// TIA Portal project "Soru9" (V15)

(* hardware
DEVICE "S7-1200 station_1"  S7-1200 Station
   slot 0: "Rack_0"  S7-1200 Rack  Rack  V1.0
   slot 1: "PLC_1"  CPU 1214C DC/DC/DC  6ES7 214-1AG40-0XB0  V4.2
*)

// ===== PLC "PLC_1"  CPU 1214C DC/DC/DC =====

VAR_GLOBAL   // PLC tag table "Default tag table"
   "Baslat" AT %I0.0 : Bool;
   "Durdur" AT %I0.1 : Bool;
   "Termik_Anahtar_Bant_1" AT %I0.2 : Bool;
   "Termik_Anahtar_Bant_2" AT %I0.3 : Bool;
   "Termik_Anahtar_Bant_3" AT %I0.4 : Bool;
   "Bant_1" AT %Q0.0 : Bool;
   "Bant_2" AT %Q0.1 : Bool;
   "Bant_3" AT %Q0.2 : Bool;
   "Aşırı_akım" AT %I0.5 : Bool;
END_VAR

// folder: System blocks/Program resources

DATA_BLOCK "Baslat_Time"   // DB2
{ S7_Optimized_Access := 'TRUE' }
AUTHOR : Simatic
FAMILY : IEC
NAME : IEC_TMR
VERSION : 1.0
// stored: InstanceOfName IEC_TIMER
"IEC_TIMER"
BEGIN
END_DATA_BLOCK

DATA_BLOCK "Dudur_Timer"   // DB3
{ S7_Optimized_Access := 'TRUE' }
AUTHOR : Simatic
FAMILY : IEC
NAME : IEC_TMR
VERSION : 1.0
// stored: InstanceOfName IEC_TIMER
"IEC_TIMER"
BEGIN
END_DATA_BLOCK

// folder: (top level)

ORGANIZATION_BLOCK "Main"   // OB1, LAD, ProgramCycle
TITLE = "Main Program Sweep (Cycle)"
{ S7_Optimized_Access := 'TRUE' }
VERSION : 0.1
   VAR_INPUT
      Initial_Call : Bool;   // Initial call of this OB
      Remanence : Bool;   // =True, if remanent data are available
   END_VAR
BEGIN

REGION Network 1: Baslama için Zaman bölümü
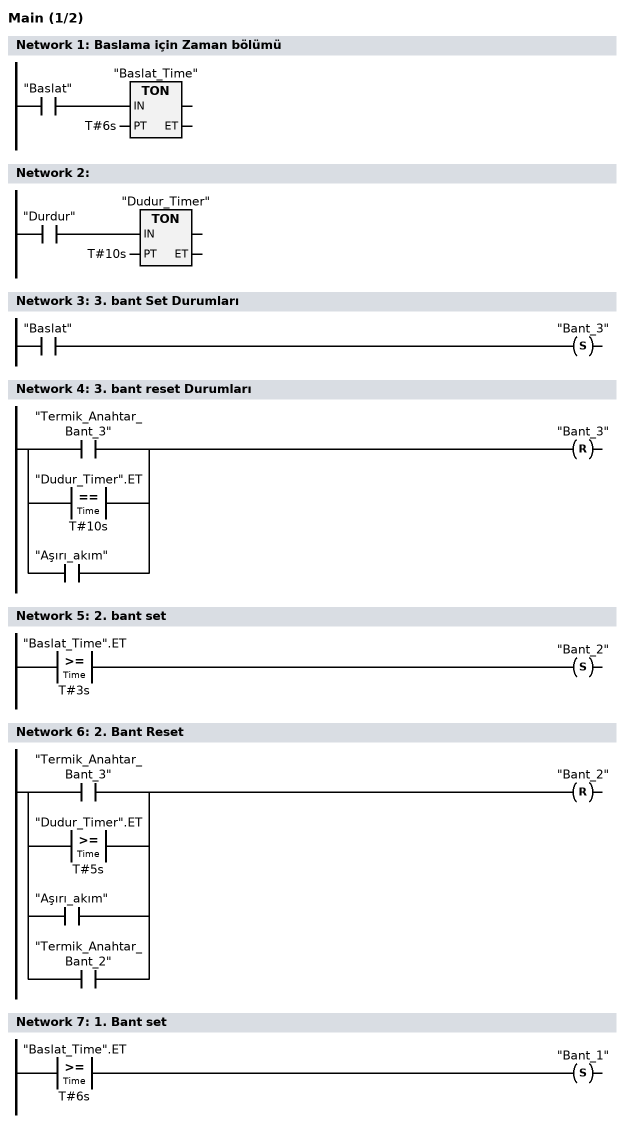
   "Baslat_Time".TON(IN := "Baslat", PT := T#6s);
END_REGION

REGION Network 2
   "Dudur_Timer".TON(IN := "Durdur", PT := T#10s);
END_REGION

REGION Network 3: 3. bant Set Durumları
   RUNG wire#powerrail
      Contact( "Baslat" )
      S_Coil( "Bant_3" )
   END_RUNG
   // the same network as SCL:
   IF "Baslat" THEN "Bant_3" := TRUE; END_IF;
END_REGION

REGION Network 4: 3. bant reset Durumları
   RUNG wire#powerrail
      Contact( "Termik_Anahtar_Bant_3" )
      wire#w1
      R_Coil( "Bant_3" )
   END_RUNG
   RUNG wire#powerrail
      { S7_Templates := "SrcType := Time" } EQ_Contact(in1 := "Dudur_Timer".ET, in2 := T#10s)
   END_RUNG wire#w1
   RUNG wire#powerrail
      Contact( "Aşırı_akım" )
   END_RUNG wire#w1
   // the same network as SCL:
   IF "Termik_Anahtar_Bant_3" OR ("Dudur_Timer".ET = T#10s) OR "Aşırı_akım" THEN "Bant_3" := FALSE; END_IF;
END_REGION

REGION Network 5: 2. bant set
   RUNG wire#powerrail
      { S7_Templates := "SrcType := Time" } GE_Contact(in1 := "Baslat_Time".ET, in2 := T#3s)
      S_Coil( "Bant_2" )
   END_RUNG
   // the same network as SCL:
   IF "Baslat_Time".ET >= T#3s THEN "Bant_2" := TRUE; END_IF;
END_REGION

REGION Network 6: 2. Bant Reset
   RUNG wire#powerrail
      Contact( "Termik_Anahtar_Bant_3" )
      wire#w1
      R_Coil( "Bant_2" )
   END_RUNG
   RUNG wire#powerrail
      { S7_Templates := "SrcType := Time" } GE_Contact(in1 := "Dudur_Timer".ET, in2 := T#5s)
   END_RUNG wire#w1
   RUNG wire#powerrail
      Contact( "Aşırı_akım" )
   END_RUNG wire#w1
   RUNG wire#powerrail
      Contact( "Termik_Anahtar_Bant_2" )
   END_RUNG wire#w1
   // the same network as SCL:
   IF "Termik_Anahtar_Bant_3" OR ("Dudur_Timer".ET >= T#5s) OR "Aşırı_akım" OR "Termik_Anahtar_Bant_2" THEN
       "Bant_2" := FALSE;
   END_IF;
END_REGION

REGION Network 7: 1. Bant set
   RUNG wire#powerrail
      { S7_Templates := "SrcType := Time" } GE_Contact(in1 := "Baslat_Time".ET, in2 := T#6s)
      S_Coil( "Bant_1" )
   END_RUNG
   // the same network as SCL:
   IF "Baslat_Time".ET >= T#6s THEN "Bant_1" := TRUE; END_IF;
END_REGION

REGION Network 8: Ban 1 Reset
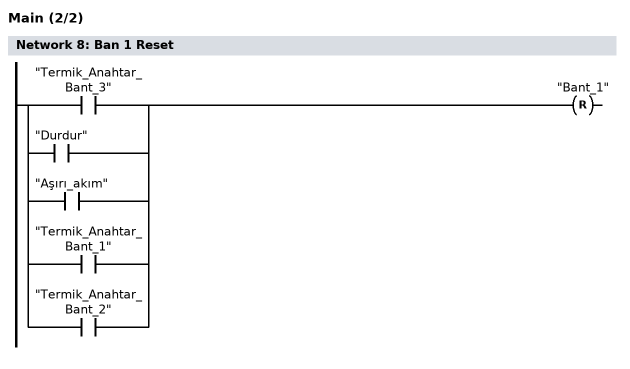
   RUNG wire#powerrail
      Contact( "Termik_Anahtar_Bant_3" )
      wire#w1
      R_Coil( "Bant_1" )
   END_RUNG
   RUNG wire#powerrail
      Contact( "Durdur" )
   END_RUNG wire#w1
   RUNG wire#powerrail
      Contact( "Aşırı_akım" )
   END_RUNG wire#w1
   RUNG wire#powerrail
      Contact( "Termik_Anahtar_Bant_1" )
   END_RUNG wire#w1
   RUNG wire#powerrail
      Contact( "Termik_Anahtar_Bant_2" )
   END_RUNG wire#w1
   // the same network as SCL:
   IF "Termik_Anahtar_Bant_3" OR "Durdur" OR "Aşırı_akım" OR "Termik_Anahtar_Bant_1" OR "Termik_Anahtar_Bant_2" THEN
       "Bant_1" := FALSE;
   END_IF;
END_REGION
END_ORGANIZATION_BLOCK